FUNCTION_BLOCK T_ComponentsIfAnyErrorReturnsErrorTrue EXTENDS T_UnitTestBase
VAR
  list : T_ComponentsCollection;
  newComponent, newComponent2 : T_ComponentMock; 
  actual1, actual2 : BOOL;
END_VAR

// Arrange
list.AddComponent(newComponent);
list.AddComponent(newComponent2);

//Act
list.CyclicLogic();
newComponent._error := TRUE;
//Assert
actual1 := list.AnyError;

assertion.AssertEquals_BOOL(TRUE, actual1, 'list.AnyError;');
TestFinished();

END_FUNCTION_BLOCK

(* stored: Version 1.1.0.1, ProductVersion 3.1.4024.12
   POU T_ComponentsIfAnyErrorReturnsErrorTrue: Id {da088fea-86d3-43fc-b325-f56f229f2fde}, SpecialFunc None *)
